TYPE dqsignal :
STRUCT
	d	:	REAL;
	q	:	REAL;
END_STRUCT
END_TYPE

(* stored: Version 1.1.0.1, ProductVersion 3.1.4022.18
   DUT dqsignal: Id {6bbdd68e-7b70-4982-b665-7e08fc0ab5ea} *)
